(* CoDeSys 2.3 export: ST_SERIAL64BYTEIN.EXP *)

(* Data type *)
TYPE ST_Serial64ByteIn :
STRUCT
	wStatus:WORD;
	aData  :ARRAY[0..63] OF BYTE;
END_STRUCT
END_TYPE
